// TIA Portal V18 export
// export: Created 2026-01-09T11:31:52.8072263Z, ExportSetting WithDefaults, DisplayName Totally Integrated Automation Portal, DisplayVersion V18 Update 5, DisplayName TIA Portal Openness, DisplayVersion V18 Update 5, DisplayName TIA Portal Teamcenter Gateway, DisplayVersion V18, DisplayName TIA Portal Version Control Interface, DisplayVersion V18, DisplayName SINAMICS Startdrive Advanced, DisplayVersion V18 SP2 Update 1, DisplayName SINAMICS Startdrive G110M, G120, G120C, G120D, G120P, G115D, DisplayVersion V18 SP2 Update 1, DisplayName SINAMICS Startdrive G130, G150, S120, S150, SINAMICS MV, S210, G220, S200, DisplayVersion V18 SP2 Update 1, DisplayName STEP 7 Professional, DisplayVersion V18 Update 5, DisplayName STEP 7 Safety, DisplayVersion V18, DisplayName WinCC Professional, DisplayVersion V18 Update 5
TagTable "Bypass"
  ST10_GeneralData_FunctionDeSelect_A_DeSelectPB_Servo380A1 : Bool  (PLC tag ST10_GeneralData.FunctionDeSelect.A.DeSelectPB_Servo380A1, CPU S71500-2PN_TP700, 1 s)
  ST10_GeneralData_FunctionDeSelect_A_FunctionDeSelected_Servo380A1 : Bool  (PLC tag ST10_GeneralData.FunctionDeSelect.A.FunctionDeSelected_Servo380A1, CPU S71500-2PN_TP700, 1 s)
  ST10_GeneralData_FunctionDeSelect_A_DeSelectPB_Servo381A1 : Bool  (PLC tag ST10_GeneralData.FunctionDeSelect.A.DeSelectPB_Servo381A1, CPU S71500-2PN_TP700, 1 s)
  ST10_GeneralData_FunctionDeSelect_A_FunctionDeSelected_Servo381A1 : Bool  (PLC tag ST10_GeneralData.FunctionDeSelect.A.FunctionDeSelected_Servo381A1, CPU S71500-2PN_TP700, 1 s)
  ST10_GeneralData_FunctionDeSelect_A_DeSelectPB_Servo383A1 : Bool  (PLC tag ST10_GeneralData.FunctionDeSelect.A.DeSelectPB_Servo383A1, CPU S71500-2PN_TP700, 1 s)
  ST10_GeneralData_FunctionDeSelect_A_FunctionDeSelected_Servo383A1 : Bool  (PLC tag ST10_GeneralData.FunctionDeSelect.A.FunctionDeSelected_Servo383A1, CPU S71500-2PN_TP700, 1 s)
  ST10_GeneralData_FunctionDeSelect_A_DeSelectPB_Reader800A1 : Bool  (PLC tag ST10_GeneralData.FunctionDeSelect.A.DeSelectPB_Reader800A1, CPU S71500-2PN_TP700, 1 s)
  ST10_GeneralData_FunctionDeSelect_A_FunctionDeSelected_Reader800A1 : Bool  (PLC tag ST10_GeneralData.FunctionDeSelect.A.FunctionDeSelected_Reader800A1, CPU S71500-2PN_TP700, 1 s)
  ST10_GeneralData_FunctionDeSelect_A_DeSelectPB_Reader801A1 : Bool  (PLC tag ST10_GeneralData.FunctionDeSelect.A.DeSelectPB_Reader801A1, CPU S71500-2PN_TP700, 1 s)
  ST10_GeneralData_FunctionDeSelect_A_FunctionDeSelected_Reader801A1 : Bool  (PLC tag ST10_GeneralData.FunctionDeSelect.A.FunctionDeSelected_Reader801A1, CPU S71500-2PN_TP700, 1 s)
  ST10_GeneralData_FunctionDeSelect_A_DeSelectPB_Reader802A1 : Bool  (PLC tag ST10_GeneralData.FunctionDeSelect.A.DeSelectPB_Reader802A1, CPU S71500-2PN_TP700, 1 s)
  ST10_GeneralData_FunctionDeSelect_A_FunctionDeSelected_Reader802A1 : Bool  (PLC tag ST10_GeneralData.FunctionDeSelect.A.FunctionDeSelected_Reader802A1, CPU S71500-2PN_TP700, 1 s)
  ST10_GeneralData_FunctionDeSelect_A_DeSelectPB_Reader803A1 : Bool  (PLC tag ST10_GeneralData.FunctionDeSelect.A.DeSelectPB_Reader803A1, CPU S71500-2PN_TP700, 1 s)
  ST10_GeneralData_FunctionDeSelect_A_FunctionDeSelected_Reader803A1 : Bool  (PLC tag ST10_GeneralData.FunctionDeSelect.A.FunctionDeSelected_Reader803A1, CPU S71500-2PN_TP700, 1 s)
  ST10_GeneralData_FunctionDeSelect_A_DeSelectPB_Reader804A1 : Bool  (PLC tag ST10_GeneralData.FunctionDeSelect.A.DeSelectPB_Reader804A1, CPU S71500-2PN_TP700, 1 s)
  ST10_GeneralData_FunctionDeSelect_A_FunctionDeSelected_Reader804A1 : Bool  (PLC tag ST10_GeneralData.FunctionDeSelect.A.FunctionDeSelected_Reader804A1, CPU S71500-2PN_TP700, 1 s)
  ST10_GeneralData_FunctionDeSelect_B_DeSelectPB_Press372A1 : Bool  (PLC tag ST10_GeneralData.FunctionDeSelect.B.DeSelectPB_Press372A1, CPU S71500-2PN_TP700, 1 s)
  ST10_GeneralData_FunctionDeSelect_B_FunctionDeSelected_Press372A1 : Bool  (PLC tag ST10_GeneralData.FunctionDeSelect.B.FunctionDeSelected_Press372A1, CPU S71500-2PN_TP700, 1 s)
  ST10_GeneralData_FunctionDeSelect_B_DeSelectPB_Press375A1 : Bool  (PLC tag ST10_GeneralData.FunctionDeSelect.B.DeSelectPB_Press375A1, CPU S71500-2PN_TP700, 1 s)
  ST10_GeneralData_FunctionDeSelect_B_FunctionDeSelected_Press375A1 : Bool  (PLC tag ST10_GeneralData.FunctionDeSelect.B.FunctionDeSelected_Press375A1, CPU S71500-2PN_TP700, 1 s)
  ST10_GeneralData_FunctionDeSelect_B_DeSelectPB_Reader806A1 : Bool  (PLC tag ST10_GeneralData.FunctionDeSelect.B.DeSelectPB_Reader806A1, CPU S71500-2PN_TP700, 1 s)
  ST10_GeneralData_FunctionDeSelect_B_FunctionDeSelected_Reader806A1 : Bool  (PLC tag ST10_GeneralData.FunctionDeSelect.B.FunctionDeSelected_Reader806A1, CPU S71500-2PN_TP700, 1 s)
  ST10_GeneralData_FunctionDeSelect_C_DeSelectPB_Servo382A1 : Bool  (PLC tag ST10_GeneralData.FunctionDeSelect.C.DeSelectPB_Servo382A1, CPU S71500-2PN_TP700, 1 s)
  ST10_GeneralData_FunctionDeSelect_C_FunctionDeSelected_Servo382A1 : Bool  (PLC tag ST10_GeneralData.FunctionDeSelect.C.FunctionDeSelected_Servo382A1, CPU S71500-2PN_TP700, 1 s)
  ST10_GeneralData_FunctionDeSelect_C_DeSelectPB_ServoIAI : Bool  (PLC tag ST10_GeneralData.FunctionDeSelect.C.DeSelectPB_ServoIAI, CPU S71500-2PN_TP700, 1 s)
  ST10_GeneralData_FunctionDeSelect_C_FunctionDeSelected_ServoIAI : Bool  (PLC tag ST10_GeneralData.FunctionDeSelect.C.FunctionDeSelected_ServoIAI, CPU S71500-2PN_TP700, 1 s)
  ST10_GeneralData_FunctionDeSelect_C_DeSelectPB_IV3810A1 : Bool  (PLC tag ST10_GeneralData.FunctionDeSelect.C.DeSelectPB_IV3810A1, CPU S71500-2PN_TP700, 1 s)
  ST10_GeneralData_FunctionDeSelect_C_FunctionDeSelected_IV3810A1 : Bool  (PLC tag ST10_GeneralData.FunctionDeSelect.C.FunctionDeSelected_IV3810A1, CPU S71500-2PN_TP700, 1 s)
  ST10_GeneralData_FunctionDeSelect_C_DeSelectPB_IV3811A1 : Bool  (PLC tag ST10_GeneralData.FunctionDeSelect.C.DeSelectPB_IV3811A1, CPU S71500-2PN_TP700, 1 s)
  ST10_GeneralData_FunctionDeSelect_C_FunctionDeSelected_IV3811A1 : Bool  (PLC tag ST10_GeneralData.FunctionDeSelect.C.FunctionDeSelected_IV3811A1, CPU S71500-2PN_TP700, 1 s)
  ST10_GeneralData_FunctionDeSelect_C_DeSelectPB_Glue : Bool  (PLC tag ST10_GeneralData.FunctionDeSelect.C.DeSelectPB_Glue, CPU S71500-2PN_TP700, 1 s)
  ST10_GeneralData_FunctionDeSelect_C_FunctionDeSelected_Glue : Bool  (PLC tag ST10_GeneralData.FunctionDeSelect.C.FunctionDeSelected_Glue, CPU S71500-2PN_TP700, 1 s)
  ST10_GeneralData_FunctionDeSelect_F_DeSelectPB_Reader805A1 : Bool  (PLC tag ST10_GeneralData.FunctionDeSelect.F.DeSelectPB_Reader805A1, CPU S71500-2PN_TP700, 1 s)
  ST10_GeneralData_FunctionDeSelect_F_FunctionDeSelected_Reader805A1 : Bool  (PLC tag ST10_GeneralData.FunctionDeSelect.F.FunctionDeSelected_Reader805A1, CPU S71500-2PN_TP700, 1 s)
  ST10_GeneralData_FunctionDeSelect_Global_DeSelectPB_DryMode : Bool  (PLC tag ST10_GeneralData.FunctionDeSelect.Global.DeSelectPB_DryMode, CPU S71500-2PN_TP700, 1 s)
  ST10_GeneralData_FunctionDeSelect_Global_FunctionDeSelected_DryMode : Bool  (PLC tag ST10_GeneralData.FunctionDeSelect.Global.FunctionDeSelected_DryMode, CPU S71500-2PN_TP700, 1 s)
  Station_Sys_Auto_Mode : Bool  (PLC tag Station_Sys.Auto.Mode, CPU S71500-2PN_TP700, 1 s)
  AutoProcessControl_C_Glue_GlueTest : Bool  (PLC tag AutoProcessControl.C_Glue.GlueTest, CPU S71500-2PN_TP700, 100 ms)
  ST10_GeneralData_FunctionDeSelect_MES_DeSelectPB : Bool  (PLC tag ST10_GeneralData.FunctionDeSelect.MES.DeSelectPB, CPU S71500-2PN_TP700, 1 s)
  ST10_GeneralData_FunctionDeSelect_MES_FunctionDeSelected : Bool  (PLC tag ST10_GeneralData.FunctionDeSelect.MES.FunctionDeSelected, CPU S71500-2PN_TP700, 1 s)
  ST10_GeneralData_FunctionDeSelect_Global_DeSelectPB_ScanFixture : Bool  (PLC tag ST10_GeneralData.FunctionDeSelect.Global.DeSelectPB_ScanFixture, CPU S71500-2PN_TP700, 1 s)
  ST10_GeneralData_FunctionDeSelect_Global_FunctionDeSelected_ScanFixture : Bool  (PLC tag ST10_GeneralData.FunctionDeSelect.Global.FunctionDeSelected_ScanFixture, CPU S71500-2PN_TP700, 1 s)
